SUBAPPLICATION TimeOutDetection (* Stand-In for the lost TimeOutDetection functionblock *)
  (* Standard: 61499-2 *)
  (* Version 0.0, 2021-07-05, Unknown, Unknown *)
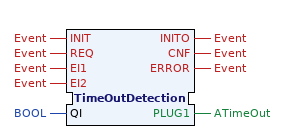
  EVENT_INPUT
    INIT; (* Initialization Request *)
    REQ; (* Normal Execution Request *)
    EI1;
    EI2;
  END_EVENT
  EVENT_OUTPUT
    INITO; (* Initialization Confirm *)
    CNF; (* Execution Confirmation *)
    ERROR;
  END_EVENT
  VAR_INPUT
    QI : BOOL; (* Input event qualifier *)
  END_VAR
  PLUGS
    PLUG1 : ATimeOut;
  END_PLUGS
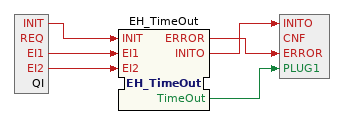
  FBS
    EH_TimeOut : EH_TimeOut;
  END_FBS
  EVENT_CONNECTIONS
    INIT TO EH_TimeOut.INIT;
    EI1 TO EH_TimeOut.EI1;
    EI2 TO EH_TimeOut.EI2;
    EH_TimeOut.ERROR TO ERROR;
    EH_TimeOut.INITO TO INITO;
  END_CONNECTIONS
  ADAPTER_CONNECTIONS
    EH_TimeOut.TimeOut TO PLUG1;
  END_CONNECTIONS
END_SUBAPPLICATION
